FUNCTION_BLOCK fbArmMoveInterLock
VAR_INPUT
	diArmPosVariable		: DINT;


END_VAR
VAR_IN_OUT

	diArmInterlock	: DINT;

END_VAR
VAR

	InterlockEn: BOOL;
END_VAR
VAR // added by the converter: edge detectors and wires of the graphical bodies
    _w1 : ANY;
END_VAR

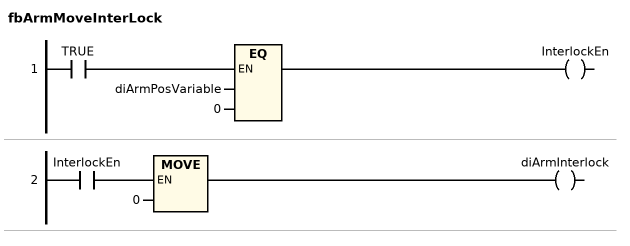
// NETWORK 1
InterlockEn := diArmPosVariable = 0;

// NETWORK 2
IF InterlockEn THEN _w1 := 0; END_IF
diArmInterlock := _w1;

END_FUNCTION_BLOCK

(* stored: Version 1.1.0.1, ProductVersion 3.1.4024.12
   POU fbArmMoveInterLock: Id {60192d24-7199-4c4a-86e2-01a3d105a4ff}, SpecialFunc None *)
